TYPE ref_sv_param :
STRUCT
	var_svType:ep_svType;
	var_mutex : INT;
	var_timeOut : TIME;
	flg_reset :BOOL;
END_STRUCT
END_TYPE

(* stored: Version 1.1.0.1, ProductVersion 3.1.4024.11
   DUT ref_sv_param: Id {9cd5e38a-e74e-44ff-aede-d46039bdd27e} *)
